ABB RobotStudio station: Trabalho Final_20220621-205907.rsstn

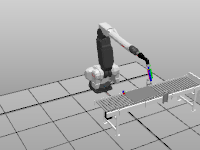
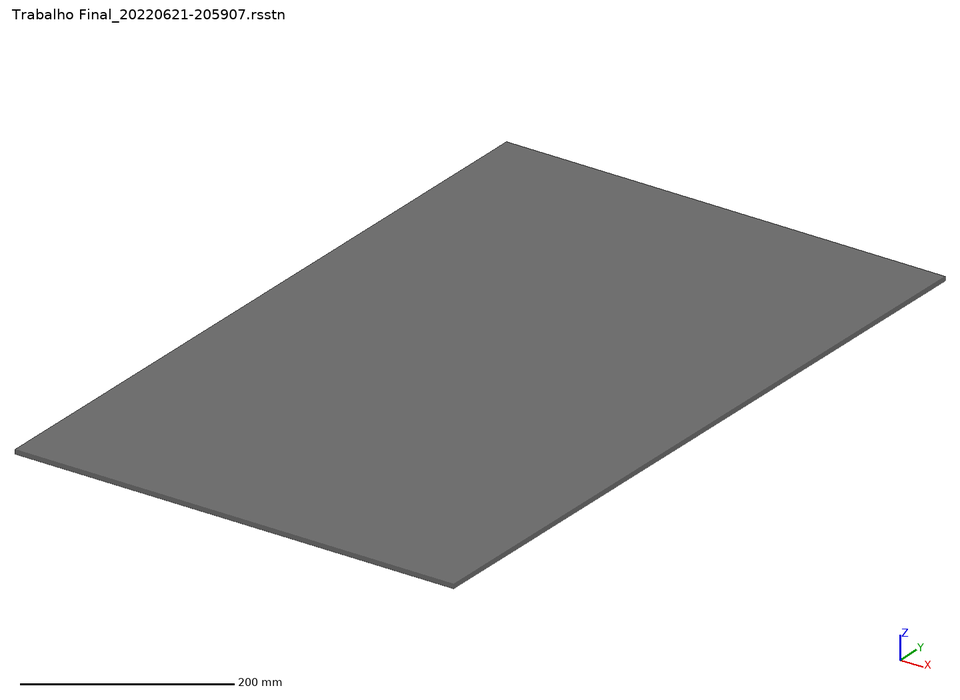
[picture v1: parts stored in the station drawn from their meshes, with robot base, taught points and paths (robot models come from the ABB library and are not in the file)]
Station Trabalho Final (saved by RobotStudio 21.4.9700.0)
Layout (positions relative to the parent item):
  - IRB5400_12_1200_1620__02 [mechanism, from Robots\IRB5400_12_1200_1620_G_02.rslib] at (0, 0, 0) mm; joint values [0.031, -0.1032, 0.1081, 0, 0, 0] (rad or m)
  - ROBOBEL926_T_TD_03 [mechanism, from Tools\ROBOBEL926_T_TD_03.rslib] at (1806.11, 55.94, 1863.79) mm, rotated rx -180 ry 83.81 rz -178.23 deg
  - 600_guide [part, from Equipment\Conveyor Guide 600.rslib] at (1788.43, 1872.85, 0) mm, rotated rx 0 ry 0 rz -90.89 deg
  - Chapa [graphiccomponentgroup]
    - Chapa [part] at (1817.02, -338.12, 823.77) mm, size 500 x 800 x 5 mm
Attachment: ROBOBEL926_T_TD_03 is attached to IRB5400_12_1200_1620__02 / Link6
Targets, tools, work objects and paths stored in the station, written as RAPID:
! task (no controller)
MODULE BASE
  TASK PERS wobjdata Chapa_Parte_Superior:=[FALSE,TRUE,"",[[1817.023,-338.123,828.769],[1,0,0,0]],[[0,0,0],[1,0,0,0]]];
ENDMODULE

! task (no controller)
MODULE CalibData
  PERS tooldata ROBOBEL926_T_TD_0:=[TRUE,[[117,0,470],[0.866025404,0,0.5,0]],[5.5,[30,0,225],[1,0,0,0],0,0,0]];
  PERS tooldata ROBOBEL926_T_TD_100:=[TRUE,[[204,0,520],[0.866025404,0,0.5,0]],[5.5,[30,0,225],[1,0,0,0],0,0,0]];
  PERS tooldata ROBOBEL926_T_TD_120:=[TRUE,[[220,0,530],[0.866025404,0,0.5,0]],[5.5,[30,0,225],[1,0,0,0],0,0,0]];
  PERS tooldata ROBOBEL926_T_TD_150:=[TRUE,[[247,0,545],[0.866025404,0,0.5,0]],[5.5,[30,0,225],[1,0,0,0],0,0,0]];
  PERS tooldata ROBOBEL926_T_TD_200:=[TRUE,[[290,0,570],[0.866025404,0,0.5,0]],[5.5,[30,0,225],[1,0,0,0],0,0,0]];
  PERS tooldata ROBOBEL926_T_TD_250:=[TRUE,[[333,0,595],[0.866025404,0,0.5,0]],[5.5,[30,0,225],[1,0,0,0],0,0,0]];
  PERS tooldata ROBOBEL926_T_TD_300:=[TRUE,[[377,0,620],[0.866025404,0,0.5,0]],[5.5,[30,0,225],[1,0,0,0],0,0,0]];
ENDMODULE

